TYPE OUT_SIGNALS :
STRUCT
	PowerError				:BOOL;
	MoveActive				:BOOL;
	MoveDone				:BOOL;
	VelocityOut				:LREAL;
	PositionOut				:LREAL;
	HaltDone				:BOOL;
	AxisCoupled				:BOOL;
	SetPosDone				:BOOL;
END_STRUCT
END_TYPE

(* stored: Version 1.1.0.1, ProductVersion 3.1.4026.12
   DUT OUT_SIGNALS: Id {2059ecb4-8f3e-47b3-b3ee-7db75fe2e3d1} *)
